SYSTEM Nutrunner
  (* Version 1.0, Author, 4DIAC-Consortium *)
  APPLICATION end2end
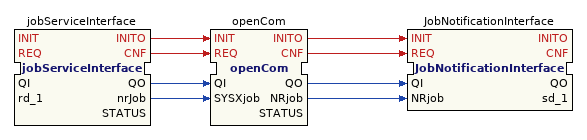
    FBS
      openCom : openCom;
      JobNotificationInterface : JobNotificationInterface;
      jobServiceInterface : jobServiceInterface;
    END_FBS
    EVENT_CONNECTIONS
      openCom.CNF TO JobNotificationInterface.REQ;
      openCom.INITO TO JobNotificationInterface.INIT;
      jobServiceInterface.INITO TO openCom.INIT;
      jobServiceInterface.CNF TO openCom.REQ;
    END_CONNECTIONS
    DATA_CONNECTIONS
      openCom.QO TO JobNotificationInterface.QI;
      openCom.NRjob TO JobNotificationInterface.NRjob;
      jobServiceInterface.QO TO openCom.QI;
      jobServiceInterface.nrJob TO openCom.SYSXjob;
    END_CONNECTIONS
  END_APPLICATION
  DEVICE FORTE_PC : FORTE_PC(MGR_ID := "localhost:61499")
    {SET_ATTRIBUTE(Profile, HOLOBLOC)}
    RESOURCE EMB_RES : EMB_RES
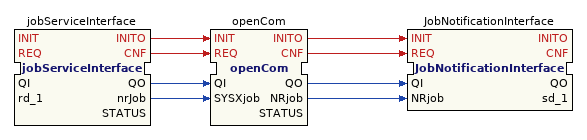
      FBS
        jobServiceInterface : jobServiceInterface;
        openCom : openCom;
        JobNotificationInterface : JobNotificationInterface;
      END_FBS
      EVENT_CONNECTIONS
        jobServiceInterface.INITO TO openCom.INIT;
        jobServiceInterface.CNF TO openCom.REQ;
        openCom.INITO TO JobNotificationInterface.INIT;
        openCom.CNF TO JobNotificationInterface.REQ;
      END_CONNECTIONS
      DATA_CONNECTIONS
        jobServiceInterface.QO TO openCom.QI;
        jobServiceInterface.nrJob TO openCom.SYSXjob;
        openCom.QO TO JobNotificationInterface.QI;
        openCom.NRjob TO JobNotificationInterface.NRjob;
      END_CONNECTIONS
    END_RESOURCE
  END_DEVICE
  MAPPINGS
    end2end.openCom ON FORTE_PC.EMB_RES.openCom;
    end2end.JobNotificationInterface ON FORTE_PC.EMB_RES.JobNotificationInterface;
    end2end.jobServiceInterface ON FORTE_PC.EMB_RES.jobServiceInterface;
  END_MAPPINGS
END_SYSTEM
